TYPE ST_StationPosition :
STRUCT
	bInit				: BOOL;
	fPositionOnTrack	: LREAL;
	nTrackId			: UINT;
	fPosition_X			: LREAL;
	fPosition_Y			: LREAL;
END_STRUCT
END_TYPE

(* stored: Version 1.1.0.1
   DUT ST_StationPosition: Id {8bd92f2b-6b4b-4688-a977-8c636394bd16} *)
